(* CODESYS project canbus.20190114.1.project

Project tree, tasks and I/O mapping:
  Changsha_Xiangji_ARM_Cortex_A9_xilinx_zynq7000_linux : Changsha Xiangji-ARM Cortex A9(xilinx zynq7000)-linux, Changsha Xiangji Hiden Technology Co.Ltd, version 3.5.10.40
    application Application
      libraries: CAA Types Extern, 3.5.10.0 (CAA Technical Workgroup); VisuDialogs, * (System); CAA Real Time Clock Extern, 3.5.10.0 (CAA Technical Workgroup); CAA Callback Extern, 3.5.11.0 (CAA Technical Workgroup); CAA Can Low Level Extern, 3.5.11.0 (CAA Technical Workgroup); CAA Can Low Level Imp Extern, 3.5.11.0 (CAA Technical Workgroup); SysMem, 3.5.12.0 (System); CAA Net Base Services, 3.5.12.0 (CAA Technical Workgroup); Standard, 3.5.12.0 (System); CAA SerialCom, 3.5.12.0 (CAA Technical Workgroup); CAA File, 3.5.12.0 (CAA Technical Workgroup); CAA DTUtil Extern, 3.5.12.0 (CAA Technical Workgroup); SysFile, 3.5.9.0 (System); SysTypes2 Interfaces, * (System)
      task VISU_TASK (cyclic, interval 100 ms, priority 31) calls VisuElems.Visu_Prg
      task task_can (cyclic, interval 50 ms, priority 5) calls prg_can0, prg_can1, prg_test_can
      CAN_COMM/
        program prg_can0 [ST]
        function CAN_Send_MSG [ST]
        program prg_can1 [ST]: can1_get_data1, can1_get_data3, can1_get_data2, can1_set_send_buf
        program prg_test_can [ST]
      visualisation main
      funcs/
    SoftMotion General Axis Pool
    IoDrvMIC7001 : IoDrvMIC7001, Cyber-MI, version 18.11.1
        unmapped channels: Ai00@C16, Ai01@C28, Ai02@C17, Ai03@C29, Ai04@C30, Ai05@C19, Ai06@C31, Ai07@C20, Ai08@C18, Ai09@D18, Ai10@D20, Ai11@D31, Ai12@D19, Ai13@D30, Ai14@D29, Ai15@D17, Ai16@D28, Ai17@D16, Ai18-Do00@C25, Ai19-Do01@C24, Ai20-Do02@C13, Ai21-Do03@C01, Ai22-Do04@C03, Ai23-Do05@C04, Ai24-Do06@C05, Ai25-Do07@C06, Ai26-Do08@C08, Ai27-Do09@C09, Ai28-Do10@C10, Ai29-Do11@C11, Ai30-Do12@D34, Ai31-Do13@D35, Ai32-Do14@D23, Ai33-Do15@D12, Ai34-Do16@D10, Ai35-Do17@D09, Ai36-Do18@D08, Ai37-Do19@D07, Ai38-Do20@D05, Ai39-Do21@D04,
          Ai40-Do22@D03, Ai41-Do23@D02, Ai42-Do24@C23, Ai43-Do25@C35, Ai44-Do26@D24, Ai45-Do27@D13, Ai46-Ao00@C22, Ai47-Ao01@D14, Ai48_Pi02, Ai49_Out5V, Ai50_VCC, Ai51_VCC_L, Ai52_VCC_R, Ai53_Pwm-i0, Ai54_Pwm-i1, Ai55_Pwm-i2, Ai56_Pwm-i3, Ai57_CPU-T, Ai58_G-x, Ai59_G-y, Ai60_G-z, Ai61-reserved, Ai62-IO-cntr, Ai63-CDS-cntr, Di00-Ai00@C16, Di01-Ai01@C28, Di02-Ai02@C17, Di03-Ai03@C29, Di04-Ai04@C30, Di05-Ai05@C19, Di06-Ai06@C31, Di07-Ai07@C20, Di08-Ai08@C18, Di09-Ai09@D18, Di10-Ai10@D20, Di11-Ai11@D31, Di12-Ai12@D19, Di13-Ai13@D30, Di14-Ai14@D29, Di15-Ai15@D17,
          Di16-Ai16@D28, Di17-Ai17@D16, Di18-Ai18@C25, Di19-Ai19@C24, Di20-Ai20@C13, Di21-Ai21@C01, Di22-Ai22@C03, Di23-Ai23@C04, Di24-Ai24@C05, Di25-Ai25@C06, Di26-Ai26@C08, Di27-Ai27@C09, Di28-Ai28@C10, Di29-Ai29@C11, Di30-Ai30@D34, Di31-Ai31@D35, Di32-Ai32@D23, Di33-Ai33@D12, Di34-Ai34@D10, Di35-Ai35@D09, Di36-Ai36@D08, Di37-Ai37@D07, Di38-Ai38@D05, Di39-Ai39@D04, Di40-Ai40@D03, Di41-Ai41@D02, Di42-Ai42@C23, Di43-Ai43@C35, Di44-Ai44@D24, Di45-Ai45@D13, Di46-Ai46@C22, Di47-Ai47@D14, Di48-Pi00@C15, Di49-Pi01@C14, Di50-Pi02@D22, Di51-Pi03@D21, Di52-reserved, Di53-reserved, Di54-reserved, Di55-reserved,
          Di56-reserved, Di57-reserved, Di58-reserved, Di59-reserved, Di60-reserved, Di61-reserved, Di62-reserved, Di63-reserved, Pi00-Di48@C15, Pi01-Di49@C14, Pi02-Di50@D22, Pi03-Di51@D21, Do00-Ai18@C25, Do01-Ai19@C24, Do02-Ai20@C13, Do03-Ai21@C01, Do04-Ai22@C03, Do05-Ai23@C04, Do06-Ai24@C05, Do07-Ai25@C06, Do08-Ai26@C08, Do09-Ai27@C09, Do10-Ai28@C10, Do11-Ai29@C11, Do12-Ai30@D34, Do13-Ai31@D35, Do14-Ai32@D23, Do15-Ai33@D12, Do16-Ai34@D10, Do17-Ai35@D09, Do18-Ai36@D08, Do19-Ai37@D07, Do20-Ai38@D05, Do21-Ai39@D04, Do22-Ai40@D03, Do23-Ai41@D02, Do24-Ai42@C23, Do25-Ai43@C35, Do26-Ai44@D24, Do27-Ai45@D13,
          Do28-Pwmi00@C33, Do29-Pwmi01@C34, Do30-Pwmi02@D25, Do31-Pwmi03@D26, PWM00@C25, PWM01@C24, PWM02@C13, PWM03@C01, PWM04@C03, PWM05@C04, PWM06@C05, PWM07@C06, PWM08@C08, PWM09@C09, PWM10@C10, PWM11@C11, PWM12@D34, PWM13@D35, PWM14@D23, PWM15@D12, PWM16@D10, PWM17@D09, PWM18@D08, PWM19@D07, PWM20@D05, PWM21@D04, PWM22@D03, PWM23@D02, PWM24@C23, PWM25@C35, PWM26@D24, PWM27@D13, PWM28-Pwmi00@C33, PWM29-Pwmi01@C34, PWM30-Pwmi02@D25, PWM31-Pwmi03@D26, PWM_I_0@C33, PWM_I_1@C34, PWM_I_2@D25, PWM_I_3@D26,
          Ao00-Ai46@C22, Ao01-Ai47@D14, LED_run, LED_err, LED_usr, ctrl_ai_raw, ctrl_adjust, ctrl_adj0, ctrl_adj1, ctrl_adj2, ctrl_adj3, ctrl_adj4
    EtherCAT_Master : EtherCAT Master, 3S - Smart Software Solutions GmbH, version 3.5.12.40
        settings: NetworkName = 'eth0'; NetworkName = "eth0"; SelectNetworkByName = True; SrcAddress1 = 8719; SrcAddress2 = 3785618642
      MIR3501 : MIR3501, Cyber-MI, order no. MIR3501, version Revision=16#00000000
          settings: CheckProductID = False; CheckVendorID = False; StationAlias = 1001; Optional = False; DeviceIdenticationADO = 0; DeviceIdenticationMode = 0; DC sync0 cycletime = 4000; DC sync1 cycletime = 4000; RxTxPdo.NumberofExcludes = 0; RxTxPdo.NumberofEntries = 24; RxTxPdo.Index = 16#1600; RxTxPdo.Fixed = True; RxTxPdo.Mandatory = True; RxTxPdo.Virtual = False; RxTxPdo.Sm = 2; RxTxPdo.Su = 2; RxTxPdo.Name = 'OUT_GENERIC process data mapping'; RxTxPdo.DependOnSlot = False; RxTxPdo.DependOnSlotGroup = False; RxTxPdo.OverwrittenByModule = False; DO-00-C01.Index = 16#7000; DO-00-C01.SubIndex = 1; DO-00-C01.Size = 1; DO-00-C01.Offset = 0; DO-00-C01.DependOnSlot = False; DO-00-C01.DependOnSlotGroup = False; DO-01-C02.Index = 16#7000; DO-01-C02.SubIndex = 2; DO-01-C02.Size = 1; DO-01-C02.Offset = 0; DO-01-C02.DependOnSlot = False; DO-01-C02.DependOnSlotGroup = False; DO-02-C03.Index = 16#7000; DO-02-C03.SubIndex = 3; DO-02-C03.Size = 1; DO-02-C03.Offset = 0; DO-02-C03.DependOnSlot = False; DO-02-C03.DependOnSlotGroup = False; DO-03-C04.Index = 16#7000; DO-03-C04.SubIndex = 4;
            DO-03-C04.Size = 1; DO-03-C04.Offset = 0; DO-03-C04.DependOnSlot = False; DO-03-C04.DependOnSlotGroup = False; DO-04-C05.Index = 16#7000; DO-04-C05.SubIndex = 5; DO-04-C05.Size = 1; DO-04-C05.Offset = 0; DO-04-C05.DependOnSlot = False; DO-04-C05.DependOnSlotGroup = False; DO-05-C06.Index = 16#7000; DO-05-C06.SubIndex = 6; DO-05-C06.Size = 1; DO-05-C06.Offset = 0; DO-05-C06.DependOnSlot = False; DO-05-C06.DependOnSlotGroup = False; DO-06-C07.Index = 16#7000; DO-06-C07.SubIndex = 7; DO-06-C07.Size = 1; DO-06-C07.Offset = 0; DO-06-C07.DependOnSlot = False; DO-06-C07.DependOnSlotGroup = False; DO-07-C08.Index = 16#7000; DO-07-C08.SubIndex = 8; DO-07-C08.Size = 1; DO-07-C08.Offset = 0; DO-07-C08.DependOnSlot = False; DO-07-C08.DependOnSlotGroup = False; DO-08-C09.Index = 16#7000; DO-08-C09.SubIndex = 9; DO-08-C09.Size = 1; DO-08-C09.Offset = 0; DO-08-C09.DependOnSlot = False; DO-08-C09.DependOnSlotGroup = False; DO-09-C10.Index = 16#7000; DO-09-C10.SubIndex = 10; DO-09-C10.Size = 1; DO-09-C10.Offset = 0; DO-09-C10.DependOnSlot = False; DO-09-C10.DependOnSlotGroup = False;
            DO-10-C11.Index = 16#7000; DO-10-C11.SubIndex = 11; DO-10-C11.Size = 1; DO-10-C11.Offset = 0; DO-10-C11.DependOnSlot = False; DO-10-C11.DependOnSlotGroup = False; DO-11-C12.Index = 16#7000; DO-11-C12.SubIndex = 12; DO-11-C12.Size = 1; DO-11-C12.Offset = 0; DO-11-C12.DependOnSlot = False; DO-11-C12.DependOnSlotGroup = False; DO-12-C26.Index = 16#7000; DO-12-C26.SubIndex = 13; DO-12-C26.Size = 1; DO-12-C26.Offset = 0; DO-12-C26.DependOnSlot = False; DO-12-C26.DependOnSlotGroup = False; DO-13-C25.Index = 16#7000; DO-13-C25.SubIndex = 14; DO-13-C25.Size = 1; DO-13-C25.Offset = 0; DO-13-C25.DependOnSlot = False; DO-13-C25.DependOnSlotGroup = False; DO-14-C34.Index = 16#7000; DO-14-C34.SubIndex = 15; DO-14-C34.Size = 1; DO-14-C34.Offset = 0; DO-14-C34.DependOnSlot = False; DO-14-C34.DependOnSlotGroup = False; DO-15-C33.Index = 16#7000; DO-15-C33.SubIndex = 16; DO-15-C33.Size = 1; DO-15-C33.Offset = 0; DO-15-C33.DependOnSlot = False; DO-15-C33.DependOnSlotGroup = False; PWM-00-C26.Index = 16#7000; PWM-00-C26.SubIndex = 17; PWM-00-C26.Size = 16; PWM-00-C26.Offset = 0;
            PWM-00-C26.DependOnSlot = False; PWM-00-C26.DependOnSlotGroup = False; PWM-01-C25.Index = 16#7000; PWM-01-C25.SubIndex = 18; PWM-01-C25.Size = 16; PWM-01-C25.Offset = 0; PWM-01-C25.DependOnSlot = False; PWM-01-C25.DependOnSlotGroup = False; PWM-02-C34.Index = 16#7000; PWM-02-C34.SubIndex = 19; PWM-02-C34.Size = 16; PWM-02-C34.Offset = 0; PWM-02-C34.DependOnSlot = False; PWM-02-C34.DependOnSlotGroup = False; PWM-03-C33.Index = 16#7000; PWM-03-C33.SubIndex = 20; PWM-03-C33.Size = 16; PWM-03-C33.Offset = 0; PWM-03-C33.DependOnSlot = False; PWM-03-C33.DependOnSlotGroup = False; PWMi-00-C26.Index = 16#7000; PWMi-00-C26.SubIndex = 21; PWMi-00-C26.Size = 16; PWMi-00-C26.Offset = 0; PWMi-00-C26.DependOnSlot = False; PWMi-00-C26.DependOnSlotGroup = False; PWMi-01-C25.Index = 16#7000; PWMi-01-C25.SubIndex = 22; PWMi-01-C25.Size = 16; PWMi-01-C25.Offset = 0; PWMi-01-C25.DependOnSlot = False; PWMi-01-C25.DependOnSlotGroup = False; PWMi-02-C34.Index = 16#7000; PWMi-02-C34.SubIndex = 23; PWMi-02-C34.Size = 16; PWMi-02-C34.Offset = 0; PWMi-02-C34.DependOnSlot = False; PWMi-02-C34.DependOnSlotGroup = False; PWMi-03-C33.Index = 16#7000; PWMi-03-C33.SubIndex = 24;
            PWMi-03-C33.Size = 16; PWMi-03-C33.Offset = 0; PWMi-03-C33.DependOnSlot = False; PWMi-03-C33.DependOnSlotGroup = False; RxTxPdo.NumberofExcludes = 0; RxTxPdo.NumberofEntries = 60; RxTxPdo.Index = 16#1A00; RxTxPdo.Fixed = True; RxTxPdo.Mandatory = True; RxTxPdo.Virtual = False; RxTxPdo.Sm = 3; RxTxPdo.Su = 3; RxTxPdo.Name = 'IN_GENERIC process data mapping'; RxTxPdo.DependOnSlot = False; RxTxPdo.DependOnSlotGroup = False; RxTxPdo.OverwrittenByModule = False; AI-00-C17.Index = 16#6000; AI-00-C17.SubIndex = 1; AI-00-C17.Size = 16; AI-00-C17.Offset = 0; AI-00-C17.DependOnSlot = False; AI-00-C17.DependOnSlotGroup = False; AI-01-C29.Index = 16#6000; AI-01-C29.SubIndex = 2; AI-01-C29.Size = 16; AI-01-C29.Offset = 0; AI-01-C29.DependOnSlot = False; AI-01-C29.DependOnSlotGroup = False; AI-02-C18.Index = 16#6000; AI-02-C18.SubIndex = 3; AI-02-C18.Size = 16; AI-02-C18.Offset = 0; AI-02-C18.DependOnSlot = False; AI-02-C18.DependOnSlotGroup = False; AI-03-C30.Index = 16#6000; AI-03-C30.SubIndex = 4; AI-03-C30.Size = 16; AI-03-C30.Offset = 0; AI-03-C30.DependOnSlot = False; AI-03-C30.DependOnSlotGroup = False;
            AI-04-C14.Index = 16#6000; AI-04-C14.SubIndex = 5; AI-04-C14.Size = 16; AI-04-C14.Offset = 0; AI-04-C14.DependOnSlot = False; AI-04-C14.DependOnSlotGroup = False; AI-05-C15.Index = 16#6000; AI-05-C15.SubIndex = 6; AI-05-C15.Size = 16; AI-05-C15.Offset = 0; AI-05-C15.DependOnSlot = False; AI-05-C15.DependOnSlotGroup = False; AI-06-C21.Index = 16#6000; AI-06-C21.SubIndex = 7; AI-06-C21.Size = 16; AI-06-C21.Offset = 0; AI-06-C21.DependOnSlot = False; AI-06-C21.DependOnSlotGroup = False; AI-07-C22.Index = 16#6000; AI-07-C22.SubIndex = 8; AI-07-C22.Size = 16; AI-07-C22.Offset = 0; AI-07-C22.DependOnSlot = False; AI-07-C22.DependOnSlotGroup = False; AI-08-C01.Index = 16#6000; AI-08-C01.SubIndex = 9; AI-08-C01.Size = 16; AI-08-C01.Offset = 0; AI-08-C01.DependOnSlot = False; AI-08-C01.DependOnSlotGroup = False; AI-09-C02.Index = 16#6000; AI-09-C02.SubIndex = 10; AI-09-C02.Size = 16; AI-09-C02.Offset = 0; AI-09-C02.DependOnSlot = False; AI-09-C02.DependOnSlotGroup = False; AI-10-C03.Index = 16#6000; AI-10-C03.SubIndex = 11; AI-10-C03.Size = 16; AI-10-C03.Offset = 0;
            AI-10-C03.DependOnSlot = False; AI-10-C03.DependOnSlotGroup = False; AI-11-C04.Index = 16#6000; AI-11-C04.SubIndex = 12; AI-11-C04.Size = 16; AI-11-C04.Offset = 0; AI-11-C04.DependOnSlot = False; AI-11-C04.DependOnSlotGroup = False; AI-12-C05.Index = 16#6000; AI-12-C05.SubIndex = 13; AI-12-C05.Size = 16; AI-12-C05.Offset = 0; AI-12-C05.DependOnSlot = False; AI-12-C05.DependOnSlotGroup = False; AI-13-C06.Index = 16#6000; AI-13-C06.SubIndex = 14; AI-13-C06.Size = 16; AI-13-C06.Offset = 0; AI-13-C06.DependOnSlot = False; AI-13-C06.DependOnSlotGroup = False; AI-14-C07.Index = 16#6000; AI-14-C07.SubIndex = 15; AI-14-C07.Size = 16; AI-14-C07.Offset = 0; AI-14-C07.DependOnSlot = False; AI-14-C07.DependOnSlotGroup = False; AI-15-C08.Index = 16#6000; AI-15-C08.SubIndex = 16; AI-15-C08.Size = 16; AI-15-C08.Offset = 0; AI-15-C08.DependOnSlot = False; AI-15-C08.DependOnSlotGroup = False; AI-16-C09.Index = 16#6000; AI-16-C09.SubIndex = 17; AI-16-C09.Size = 16; AI-16-C09.Offset = 0; AI-16-C09.DependOnSlot = False; AI-16-C09.DependOnSlotGroup = False; AI-17-C10.Index = 16#6000; AI-17-C10.SubIndex = 18;
            AI-17-C10.Size = 16; AI-17-C10.Offset = 0; AI-17-C10.DependOnSlot = False; AI-17-C10.DependOnSlotGroup = False; AI-18-C11.Index = 16#6000; AI-18-C11.SubIndex = 19; AI-18-C11.Size = 16; AI-18-C11.Offset = 0; AI-18-C11.DependOnSlot = False; AI-18-C11.DependOnSlotGroup = False; AI-19-C12.Index = 16#6000; AI-19-C12.SubIndex = 20; AI-19-C12.Size = 16; AI-19-C12.Offset = 0; AI-19-C12.DependOnSlot = False; AI-19-C12.DependOnSlotGroup = False; AI-20.Index = 16#6000; AI-20.SubIndex = 21; AI-20.Size = 16; AI-20.Offset = 0; AI-20.DependOnSlot = False; AI-20.DependOnSlotGroup = False; AI-21.Index = 16#6000; AI-21.SubIndex = 22; AI-21.Size = 16; AI-21.Offset = 0; AI-21.DependOnSlot = False; AI-21.DependOnSlotGroup = False; AI-22.Index = 16#6000; AI-22.SubIndex = 23; AI-22.Size = 16; AI-22.Offset = 0; AI-22.DependOnSlot = False; AI-22.DependOnSlotGroup = False; AI-23.Index = 16#6000; AI-23.SubIndex = 24; AI-23.Size = 16; AI-23.Offset = 0; AI-23.DependOnSlot = False; AI-23.DependOnSlotGroup = False;
            DI-00-C17.Index = 16#6000; DI-00-C17.SubIndex = 25; DI-00-C17.Size = 1; DI-00-C17.Offset = 0; DI-00-C17.DependOnSlot = False; DI-00-C17.DependOnSlotGroup = False; DI-01-C29.Index = 16#6000; DI-01-C29.SubIndex = 26; DI-01-C29.Size = 1; DI-01-C29.Offset = 0; DI-01-C29.DependOnSlot = False; DI-01-C29.DependOnSlotGroup = False; DI-02-C18.Index = 16#6000; DI-02-C18.SubIndex = 27; DI-02-C18.Size = 1; DI-02-C18.Offset = 0; DI-02-C18.DependOnSlot = False; DI-02-C18.DependOnSlotGroup = False; DI-03-C30.Index = 16#6000; DI-03-C30.SubIndex = 28; DI-03-C30.Size = 1; DI-03-C30.Offset = 0; DI-03-C30.DependOnSlot = False; DI-03-C30.DependOnSlotGroup = False; DI-04-C14.Index = 16#6000; DI-04-C14.SubIndex = 29; DI-04-C14.Size = 1; DI-04-C14.Offset = 0; DI-04-C14.DependOnSlot = False; DI-04-C14.DependOnSlotGroup = False; DI-05-C15.Index = 16#6000; DI-05-C15.SubIndex = 30; DI-05-C15.Size = 1; DI-05-C15.Offset = 0; DI-05-C15.DependOnSlot = False; DI-05-C15.DependOnSlotGroup = False; DI-06-C21.Index = 16#6000; DI-06-C21.SubIndex = 31; DI-06-C21.Size = 1; DI-06-C21.Offset = 0;
            DI-06-C21.DependOnSlot = False; DI-06-C21.DependOnSlotGroup = False; DI-07-C22.Index = 16#6000; DI-07-C22.SubIndex = 32; DI-07-C22.Size = 1; DI-07-C22.Offset = 0; DI-07-C22.DependOnSlot = False; DI-07-C22.DependOnSlotGroup = False; DI-08-C01.Index = 16#6000; DI-08-C01.SubIndex = 33; DI-08-C01.Size = 1; DI-08-C01.Offset = 0; DI-08-C01.DependOnSlot = False; DI-08-C01.DependOnSlotGroup = False; DI-09-C02.Index = 16#6000; DI-09-C02.SubIndex = 34; DI-09-C02.Size = 1; DI-09-C02.Offset = 0; DI-09-C02.DependOnSlot = False; DI-09-C02.DependOnSlotGroup = False; DI-10-C03.Index = 16#6000; DI-10-C03.SubIndex = 35; DI-10-C03.Size = 1; DI-10-C03.Offset = 0; DI-10-C03.DependOnSlot = False; DI-10-C03.DependOnSlotGroup = False; DI-11-C04.Index = 16#6000; DI-11-C04.SubIndex = 36; DI-11-C04.Size = 1; DI-11-C04.Offset = 0; DI-11-C04.DependOnSlot = False; DI-11-C04.DependOnSlotGroup = False; DI-12-C05.Index = 16#6000; DI-12-C05.SubIndex = 37; DI-12-C05.Size = 1; DI-12-C05.Offset = 0; DI-12-C05.DependOnSlot = False; DI-12-C05.DependOnSlotGroup = False; DI-13-C06.Index = 16#6000; DI-13-C06.SubIndex = 38;
            DI-13-C06.Size = 1; DI-13-C06.Offset = 0; DI-13-C06.DependOnSlot = False; DI-13-C06.DependOnSlotGroup = False; DI-14-C07.Index = 16#6000; DI-14-C07.SubIndex = 39; DI-14-C07.Size = 1; DI-14-C07.Offset = 0; DI-14-C07.DependOnSlot = False; DI-14-C07.DependOnSlotGroup = False; DI-15-C08.Index = 16#6000; DI-15-C08.SubIndex = 40; DI-15-C08.Size = 1; DI-15-C08.Offset = 0; DI-15-C08.DependOnSlot = False; DI-15-C08.DependOnSlotGroup = False; DI-16-C09.Index = 16#6000; DI-16-C09.SubIndex = 41; DI-16-C09.Size = 1; DI-16-C09.Offset = 0; DI-16-C09.DependOnSlot = False; DI-16-C09.DependOnSlotGroup = False; DI-17-C10.Index = 16#6000; DI-17-C10.SubIndex = 42; DI-17-C10.Size = 1; DI-17-C10.Offset = 0; DI-17-C10.DependOnSlot = False; DI-17-C10.DependOnSlotGroup = False; DI-18-C11.Index = 16#6000; DI-18-C11.SubIndex = 43; DI-18-C11.Size = 1; DI-18-C11.Offset = 0; DI-18-C11.DependOnSlot = False; DI-18-C11.DependOnSlotGroup = False; DI-19-C12.Index = 16#6000; DI-19-C12.SubIndex = 44; DI-19-C12.Size = 1; DI-19-C12.Offset = 0; DI-19-C12.DependOnSlot = False; DI-19-C12.DependOnSlotGroup = False;
            DI-20-C27.Index = 16#6000; DI-20-C27.SubIndex = 45; DI-20-C27.Size = 1; DI-20-C27.Offset = 0; DI-20-C27.DependOnSlot = False; DI-20-C27.DependOnSlotGroup = False; DI-21-C16.Index = 16#6000; DI-21-C16.SubIndex = 46; DI-21-C16.Size = 1; DI-21-C16.Offset = 0; DI-21-C16.DependOnSlot = False; DI-21-C16.DependOnSlotGroup = False; DI-22-C19.Index = 16#6000; DI-22-C19.SubIndex = 47; DI-22-C19.Size = 1; DI-22-C19.Offset = 0; DI-22-C19.DependOnSlot = False; DI-22-C19.DependOnSlotGroup = False; DI-23-C20.Index = 16#6000; DI-23-C20.SubIndex = 48; DI-23-C20.Size = 1; DI-23-C20.Offset = 0; DI-23-C20.DependOnSlot = False; DI-23-C20.DependOnSlotGroup = False; DI-24.Index = 16#6000; DI-24.SubIndex = 49; DI-24.Size = 1; DI-24.Offset = 0; DI-24.DependOnSlot = False; DI-24.DependOnSlotGroup = False; DI-25.Index = 16#6000; DI-25.SubIndex = 50; DI-25.Size = 1; DI-25.Offset = 0; DI-25.DependOnSlot = False; DI-25.DependOnSlotGroup = False; DI-26.Index = 16#6000; DI-26.SubIndex = 51; DI-26.Size = 1; DI-26.Offset = 0;
            DI-26.DependOnSlot = False; DI-26.DependOnSlotGroup = False; DI-27.Index = 16#6000; DI-27.SubIndex = 52; DI-27.Size = 1; DI-27.Offset = 0; DI-27.DependOnSlot = False; DI-27.DependOnSlotGroup = False; DI-28.Index = 16#6000; DI-28.SubIndex = 53; DI-28.Size = 1; DI-28.Offset = 0; DI-28.DependOnSlot = False; DI-28.DependOnSlotGroup = False; DI-29.Index = 16#6000; DI-29.SubIndex = 54; DI-29.Size = 1; DI-29.Offset = 0; DI-29.DependOnSlot = False; DI-29.DependOnSlotGroup = False; DI-30.Index = 16#6000; DI-30.SubIndex = 55; DI-30.Size = 1; DI-30.Offset = 0; DI-30.DependOnSlot = False; DI-30.DependOnSlotGroup = False; DI-31.Index = 16#6000; DI-31.SubIndex = 56; DI-31.Size = 1; DI-31.Offset = 0; DI-31.DependOnSlot = False; DI-31.DependOnSlotGroup = False; PI-00-C27.Index = 16#6000; PI-00-C27.SubIndex = 57; PI-00-C27.Size = 16; PI-00-C27.Offset = 0; PI-00-C27.DependOnSlot = False; PI-00-C27.DependOnSlotGroup = False; PI-01-C16.Index = 16#6000; PI-01-C16.SubIndex = 58;
            PI-01-C16.Size = 16; PI-01-C16.Offset = 0; PI-01-C16.DependOnSlot = False; PI-01-C16.DependOnSlotGroup = False; PI-02-C19.Index = 16#6000; PI-02-C19.SubIndex = 59; PI-02-C19.Size = 16; PI-02-C19.Offset = 0; PI-02-C19.DependOnSlot = False; PI-02-C19.DependOnSlotGroup = False; PI-03-C20.Index = 16#6000; PI-03-C20.SubIndex = 60; PI-03-C20.Size = 16; PI-03-C20.Offset = 0; PI-03-C20.DependOnSlot = False; PI-03-C20.DependOnSlotGroup = False; DO-00-C01.Name = 'DO-00-C01'; DO-00-C01.DataType = 'BIT'; DO-00-C01.Default = ''; DO-00-C01.Comment = ''; DO-01-C02.Name = 'DO-01-C02'; DO-01-C02.DataType = 'BIT'; DO-01-C02.Default = ''; DO-01-C02.Comment = ''; DO-02-C03.Name = 'DO-02-C03'; DO-02-C03.DataType = 'BIT'; DO-02-C03.Default = ''; DO-02-C03.Comment = ''; DO-03-C04.Name = 'DO-03-C04'; DO-03-C04.DataType = 'BIT'; DO-03-C04.Default = ''; DO-03-C04.Comment = ''; DO-04-C05.Name = 'DO-04-C05'; DO-04-C05.DataType = 'BIT'; DO-04-C05.Default = ''; DO-04-C05.Comment = ''; DO-05-C06.Name = 'DO-05-C06'; DO-05-C06.DataType = 'BIT'; DO-05-C06.Default = ''; DO-05-C06.Comment = '';
            DO-06-C07.Name = 'DO-06-C07'; DO-06-C07.DataType = 'BIT'; DO-06-C07.Default = ''; DO-06-C07.Comment = ''; DO-07-C08.Name = 'DO-07-C08'; DO-07-C08.DataType = 'BIT'; DO-07-C08.Default = ''; DO-07-C08.Comment = ''; DO-08-C09.Name = 'DO-08-C09'; DO-08-C09.DataType = 'BIT'; DO-08-C09.Default = ''; DO-08-C09.Comment = ''; DO-09-C10.Name = 'DO-09-C10'; DO-09-C10.DataType = 'BIT'; DO-09-C10.Default = ''; DO-09-C10.Comment = ''; DO-10-C11.Name = 'DO-10-C11'; DO-10-C11.DataType = 'BIT'; DO-10-C11.Default = ''; DO-10-C11.Comment = ''; DO-11-C12.Name = 'DO-11-C12'; DO-11-C12.DataType = 'BIT'; DO-11-C12.Default = ''; DO-11-C12.Comment = ''; DO-12-C26.Name = 'DO-12-C26'; DO-12-C26.DataType = 'BIT'; DO-12-C26.Default = ''; DO-12-C26.Comment = ''; DO-13-C25.Name = 'DO-13-C25'; DO-13-C25.DataType = 'BIT'; DO-13-C25.Default = ''; DO-13-C25.Comment = ''; DO-14-C34.Name = 'DO-14-C34'; DO-14-C34.DataType = 'BIT'; DO-14-C34.Default = ''; DO-14-C34.Comment = ''; DO-15-C33.Name = 'DO-15-C33'; DO-15-C33.DataType = 'BIT'; DO-15-C33.Default = ''; DO-15-C33.Comment = '';
            PWM-00-C26.Name = 'PWM-00-C26'; PWM-00-C26.DataType = 'UINT'; PWM-00-C26.Default = ''; PWM-00-C26.Comment = ''; PWM-01-C25.Name = 'PWM-01-C25'; PWM-01-C25.DataType = 'UINT'; PWM-01-C25.Default = ''; PWM-01-C25.Comment = ''; PWM-02-C34.Name = 'PWM-02-C34'; PWM-02-C34.DataType = 'UINT'; PWM-02-C34.Default = ''; PWM-02-C34.Comment = ''; PWM-03-C33.Name = 'PWM-03-C33'; PWM-03-C33.DataType = 'UINT'; PWM-03-C33.Default = ''; PWM-03-C33.Comment = ''; PWMi-00-C26.Name = 'PWMi-00-C26'; PWMi-00-C26.DataType = 'UINT'; PWMi-00-C26.Default = ''; PWMi-00-C26.Comment = ''; PWMi-01-C25.Name = 'PWMi-01-C25'; PWMi-01-C25.DataType = 'UINT'; PWMi-01-C25.Default = ''; PWMi-01-C25.Comment = ''; PWMi-02-C34.Name = 'PWMi-02-C34'; PWMi-02-C34.DataType = 'UINT'; PWMi-02-C34.Default = ''; PWMi-02-C34.Comment = ''; PWMi-03-C33.Name = 'PWMi-03-C33'; PWMi-03-C33.DataType = 'UINT'; PWMi-03-C33.Default = ''; PWMi-03-C33.Comment = ''; AI-00-C17.Name = 'AI-00-C17'; AI-00-C17.DataType = 'UINT'; AI-00-C17.Default = ''; AI-00-C17.Comment = ''; AI-01-C29.Name = 'AI-01-C29'; AI-01-C29.DataType = 'UINT'; AI-01-C29.Default = ''; AI-01-C29.Comment = '';
            AI-02-C18.Name = 'AI-02-C18'; AI-02-C18.DataType = 'UINT'; AI-02-C18.Default = ''; AI-02-C18.Comment = ''; AI-03-C30.Name = 'AI-03-C30'; AI-03-C30.DataType = 'UINT'; AI-03-C30.Default = ''; AI-03-C30.Comment = ''; AI-04-C14.Name = 'AI-04-C14'; AI-04-C14.DataType = 'UINT'; AI-04-C14.Default = ''; AI-04-C14.Comment = ''; AI-05-C15.Name = 'AI-05-C15'; AI-05-C15.DataType = 'UINT'; AI-05-C15.Default = ''; AI-05-C15.Comment = ''; AI-06-C21.Name = 'AI-06-C21'; AI-06-C21.DataType = 'UINT'; AI-06-C21.Default = ''; AI-06-C21.Comment = ''; AI-07-C22.Name = 'AI-07-C22'; AI-07-C22.DataType = 'UINT'; AI-07-C22.Default = ''; AI-07-C22.Comment = ''; AI-08-C01.Name = 'AI-08-C01'; AI-08-C01.DataType = 'UINT'; AI-08-C01.Default = ''; AI-08-C01.Comment = ''; AI-09-C02.Name = 'AI-09-C02'; AI-09-C02.DataType = 'UINT'; AI-09-C02.Default = ''; AI-09-C02.Comment = ''; AI-10-C03.Name = 'AI-10-C03'; AI-10-C03.DataType = 'UINT'; AI-10-C03.Default = ''; AI-10-C03.Comment = ''; AI-11-C04.Name = 'AI-11-C04'; AI-11-C04.DataType = 'UINT'; AI-11-C04.Default = ''; AI-11-C04.Comment = '';
            AI-12-C05.Name = 'AI-12-C05'; AI-12-C05.DataType = 'UINT'; AI-12-C05.Default = ''; AI-12-C05.Comment = ''; AI-13-C06.Name = 'AI-13-C06'; AI-13-C06.DataType = 'UINT'; AI-13-C06.Default = ''; AI-13-C06.Comment = ''; AI-14-C07.Name = 'AI-14-C07'; AI-14-C07.DataType = 'UINT'; AI-14-C07.Default = ''; AI-14-C07.Comment = ''; AI-15-C08.Name = 'AI-15-C08'; AI-15-C08.DataType = 'UINT'; AI-15-C08.Default = ''; AI-15-C08.Comment = ''; AI-16-C09.Name = 'AI-16-C09'; AI-16-C09.DataType = 'UINT'; AI-16-C09.Default = ''; AI-16-C09.Comment = ''; AI-17-C10.Name = 'AI-17-C10'; AI-17-C10.DataType = 'UINT'; AI-17-C10.Default = ''; AI-17-C10.Comment = ''; AI-18-C11.Name = 'AI-18-C11'; AI-18-C11.DataType = 'UINT'; AI-18-C11.Default = ''; AI-18-C11.Comment = ''; AI-19-C12.Name = 'AI-19-C12'; AI-19-C12.DataType = 'UINT'; AI-19-C12.Default = ''; AI-19-C12.Comment = ''; AI-20.Name = 'AI-20'; AI-20.DataType = 'UINT'; AI-20.Default = ''; AI-20.Comment = ''; AI-21.Name = 'AI-21'; AI-21.DataType = 'UINT'; AI-21.Default = ''; AI-21.Comment = '';
            AI-22.Name = 'AI-22'; AI-22.DataType = 'UINT'; AI-22.Default = ''; AI-22.Comment = ''; AI-23.Name = 'AI-23'; AI-23.DataType = 'UINT'; AI-23.Default = ''; AI-23.Comment = ''; DI-00-C17.Name = 'DI-00-C17'; DI-00-C17.DataType = 'BIT'; DI-00-C17.Default = ''; DI-00-C17.Comment = ''; DI-01-C29.Name = 'DI-01-C29'; DI-01-C29.DataType = 'BIT'; DI-01-C29.Default = ''; DI-01-C29.Comment = ''; DI-02-C18.Name = 'DI-02-C18'; DI-02-C18.DataType = 'BIT'; DI-02-C18.Default = ''; DI-02-C18.Comment = ''; DI-03-C30.Name = 'DI-03-C30'; DI-03-C30.DataType = 'BIT'; DI-03-C30.Default = ''; DI-03-C30.Comment = ''; DI-04-C14.Name = 'DI-04-C14'; DI-04-C14.DataType = 'BIT'; DI-04-C14.Default = ''; DI-04-C14.Comment = ''; DI-05-C15.Name = 'DI-05-C15'; DI-05-C15.DataType = 'BIT'; DI-05-C15.Default = ''; DI-05-C15.Comment = ''; DI-06-C21.Name = 'DI-06-C21'; DI-06-C21.DataType = 'BIT'; DI-06-C21.Default = ''; DI-06-C21.Comment = ''; DI-07-C22.Name = 'DI-07-C22'; DI-07-C22.DataType = 'BIT'; DI-07-C22.Default = ''; DI-07-C22.Comment = '';
            DI-08-C01.Name = 'DI-08-C01'; DI-08-C01.DataType = 'BIT'; DI-08-C01.Default = ''; DI-08-C01.Comment = ''; DI-09-C02.Name = 'DI-09-C02'; DI-09-C02.DataType = 'BIT'; DI-09-C02.Default = ''; DI-09-C02.Comment = ''; DI-10-C03.Name = 'DI-10-C03'; DI-10-C03.DataType = 'BIT'; DI-10-C03.Default = ''; DI-10-C03.Comment = ''; DI-11-C04.Name = 'DI-11-C04'; DI-11-C04.DataType = 'BIT'; DI-11-C04.Default = ''; DI-11-C04.Comment = ''; DI-12-C05.Name = 'DI-12-C05'; DI-12-C05.DataType = 'BIT'; DI-12-C05.Default = ''; DI-12-C05.Comment = ''; DI-13-C06.Name = 'DI-13-C06'; DI-13-C06.DataType = 'BIT'; DI-13-C06.Default = ''; DI-13-C06.Comment = ''; DI-14-C07.Name = 'DI-14-C07'; DI-14-C07.DataType = 'BIT'; DI-14-C07.Default = ''; DI-14-C07.Comment = ''; DI-15-C08.Name = 'DI-15-C08'; DI-15-C08.DataType = 'BIT'; DI-15-C08.Default = ''; DI-15-C08.Comment = ''; DI-16-C09.Name = 'DI-16-C09'; DI-16-C09.DataType = 'BIT'; DI-16-C09.Default = ''; DI-16-C09.Comment = ''; DI-17-C10.Name = 'DI-17-C10'; DI-17-C10.DataType = 'BIT'; DI-17-C10.Default = ''; DI-17-C10.Comment = '';
            DI-18-C11.Name = 'DI-18-C11'; DI-18-C11.DataType = 'BIT'; DI-18-C11.Default = ''; DI-18-C11.Comment = ''; DI-19-C12.Name = 'DI-19-C12'; DI-19-C12.DataType = 'BIT'; DI-19-C12.Default = ''; DI-19-C12.Comment = ''; DI-20-C27.Name = 'DI-20-C27'; DI-20-C27.DataType = 'BIT'; DI-20-C27.Default = ''; DI-20-C27.Comment = ''; DI-21-C16.Name = 'DI-21-C16'; DI-21-C16.DataType = 'BIT'; DI-21-C16.Default = ''; DI-21-C16.Comment = ''; DI-22-C19.Name = 'DI-22-C19'; DI-22-C19.DataType = 'BIT'; DI-22-C19.Default = ''; DI-22-C19.Comment = ''; DI-23-C20.Name = 'DI-23-C20'; DI-23-C20.DataType = 'BIT'; DI-23-C20.Default = ''; DI-23-C20.Comment = ''; DI-24.Name = 'DI-24'; DI-24.DataType = 'BIT'; DI-24.Default = ''; DI-24.Comment = ''; DI-25.Name = 'DI-25'; DI-25.DataType = 'BIT'; DI-25.Default = ''; DI-25.Comment = ''; DI-26.Name = 'DI-26'; DI-26.DataType = 'BIT'; DI-26.Default = ''; DI-26.Comment = ''; DI-27.Name = 'DI-27'; DI-27.DataType = 'BIT'; DI-27.Default = ''; DI-27.Comment = '';
            DI-28.Name = 'DI-28'; DI-28.DataType = 'BIT'; DI-28.Default = ''; DI-28.Comment = ''; DI-29.Name = 'DI-29'; DI-29.DataType = 'BIT'; DI-29.Default = ''; DI-29.Comment = ''; DI-30.Name = 'DI-30'; DI-30.DataType = 'BIT'; DI-30.Default = ''; DI-30.Comment = ''; DI-31.Name = 'DI-31'; DI-31.DataType = 'BIT'; DI-31.Default = ''; DI-31.Comment = ''; PI-00-C27.Name = 'PI-00-C27'; PI-00-C27.DataType = 'UINT'; PI-00-C27.Default = ''; PI-00-C27.Comment = ''; PI-01-C16.Name = 'PI-01-C16'; PI-01-C16.DataType = 'UINT'; PI-01-C16.Default = ''; PI-01-C16.Comment = ''; PI-02-C19.Name = 'PI-02-C19'; PI-02-C19.DataType = 'UINT'; PI-02-C19.Default = ''; PI-02-C19.Comment = ''; PI-03-C20.Name = 'PI-03-C20'; PI-03-C20.DataType = 'UINT'; PI-03-C20.Default = ''; PI-03-C20.Comment = ''
          unmapped channels: DO-00-C01, DO-01-C02, DO-02-C03, DO-03-C04, DO-04-C05, DO-05-C06, DO-06-C07, DO-07-C08, DO-08-C09, DO-09-C10, DO-10-C11, DO-11-C12, DO-12-C26, DO-13-C25, DO-14-C34, DO-15-C33, PWM-00-C26, PWM-01-C25, PWM-02-C34, PWM-03-C33, PWMi-00-C26, PWMi-01-C25, PWMi-02-C34, PWMi-03-C33, AI-00-C17, AI-01-C29, AI-02-C18, AI-03-C30, AI-04-C14, AI-05-C15, AI-06-C21, AI-07-C22, AI-08-C01, AI-09-C02, AI-10-C03, AI-11-C04, AI-12-C05, AI-13-C06, AI-14-C07, AI-15-C08,
            AI-16-C09, AI-17-C10, AI-18-C11, AI-19-C12, AI-20, AI-21, AI-22, AI-23, DI-00-C17, DI-01-C29, DI-02-C18, DI-03-C30, DI-04-C14, DI-05-C15, DI-06-C21, DI-07-C22, DI-08-C01, DI-09-C02, DI-10-C03, DI-11-C04, DI-12-C05, DI-13-C06, DI-14-C07, DI-15-C08, DI-16-C09, DI-17-C10, DI-18-C11, DI-19-C12, DI-20-C27, DI-21-C16, DI-22-C19, DI-23-C20, DI-24, DI-25, DI-26, DI-27, DI-28, DI-29, DI-30, DI-31,
            PI-00-C27, PI-01-C16, PI-02-C19, PI-03-C20
  5ce3da45-db07-42e7-a21c-a00fff4ed8f6|C:\Users\Administrator\Desktop\robotview1.bmp
  5ce3da45-db07-42e7-a21c-a00fff4ed8f6|C:\Users\Administrator\Desktop\robotview2.bmp
  text list GlobalTextList
  5ce3da45-db07-42e7-a21c-a00fff4ed8f6|C:\Users\Administrator\Desktop\1129.bmp
  5ce3da45-db07-42e7-a21c-a00fff4ed8f6|C:\Users\Administrator\Desktop\robotview0.bmp
*)

// Changsha_Xiangji_ARM_Cortex_A9_xilinx_zynq7000_linux/Application/CAN_COMM/prg_can0
PROGRAM prg_can0   //CAN0   与底盘和显示屏通信
VAR
	hCan0:CAA.HANDLE:=0;
    CanWriteData : ARRAY[0..7] OF BYTE;
    CanWriteMsgID:UDINT;
	CanReadData : ARRAY[0..7] OF BYTE;  
	CanReadMsgID:UDINT;
	bModifyTimeFlag :BOOL := FALSE;
	
	//通过CAN总线从底盘读到的信息
	can_data_ready:BOOL := FALSE;
	can_data_speed:BYTE := 0;
	can_data_soc:BYTE := 0;
	
	//通过CAN总线从显示屏读到的信息
	c00byte0bit0_both_wash_sweep:BOOL := FALSE;
	c00byte0bit1_left_wash_sweep:BOOL := FALSE;
	c00byte0bit2_right_wash_sweep:BOOL := FALSE;
	c00byte0bit3_both_sweep:BOOL := FALSE;
	c00byte0bit4_left_sweep:BOOL := FALSE;
	c00byte0bit5_right_sweep:BOOL := FALSE;
	c00byte0bit6_both_wash:BOOL := FALSE;
	c00byte0bit7_left_wash:BOOL := FALSE;
	
	c00byte1bit0_right_wash:BOOL := FALSE;
	c00byte1bit1_stop_sweep:BOOL := FALSE;
	c00byte1bit2_start_motor:BOOL := FALSE;
	c00byte1bit3_stop_motor:BOOL := FALSE;
	c00byte1bit4_speed_add:BOOL := FALSE;
	c00byte1bit5_speed_dec:BOOL := FALSE;
	c00byte1bit6_normal_speed:BOOL := FALSE;
	c00byte1bit7_high_speed:BOOL := FALSE;
	
	c00byte2bit0_garbage_close:BOOL := FALSE;
	c00byte2bit1_garbage_open:BOOL := FALSE;
	c00byte2bit2_garbage_up:BOOL := FALSE;
	c00byte2bit3_garbage_down:BOOL := FALSE;
	c00byte2bit4_fog_bump:BOOL := FALSE;
	c00byte2bit5_selfclean:BOOL := FALSE;
	c00byte2bit6_wastewater_pump:BOOL := FALSE;
	c00byte2bit7_res :BOOL := FALSE;
	
	c00byte3bit0_sweep_high:BOOL := FALSE;
	c00byte3bit1_sweep_middle:BOOL := FALSE;
	c00byte3bit2_sweep_low:BOOL := FALSE;
	c00byte3bit3_highpress_wash:BOOL := FALSE;
	c00byte3bit4_pointshoot_up:BOOL := FALSE;
	c00byte3bit5_pointshoot_down:BOOL := FALSE;
	c00byte3bit6_pointshoot_left:BOOL := FALSE;
	c00byte3bit7_pointshoot_right:BOOL := FALSE;

	c00byte4bit0_drain_start:BOOL := FALSE;
	c00byte4bit1_drain_auto:BOOL := FALSE;
	c00byte4bit2_drain_manual:BOOL := FALSE;
	c00byte4bit3_left_drain:BOOL := FALSE;
	c00byte4bit4_right_drain:BOOL := FALSE;
	c00byte4bit5_sub_drain:BOOL := FALSE;
	c00byte4bit6_selfclean_drain:BOOL := FALSE;
	c00byte4bit7_spout_drain:BOOL := FALSE;
	
	c00byte6bit0_func_test:BOOL := FALSE;
	c00byte6bit1_change_sweeper:BOOL := FALSE;
	c00byte6bit2_intelligent:BOOL := FALSE;
	c00byte6bit3_cleanly:BOOL := FALSE;
	c00byte6bit4_normal:BOOL := FALSE;
	c00byte6bit5_dirty:BOOL := FALSE;
	
	c01byte0bit3_test_watercooler_pump:BOOL := FALSE;
	c01byte0bit4_test_cooler_fan:BOOL := FALSE;
	
	c01byte1bit0_test_sweeper_middle:BOOL := FALSE;
	c01byte1bit1_test_sweeper_low:BOOL := FALSE;
	c01byte1bit2_test_left_sweeper:BOOL := FALSE;
	c01byte1bit3_test_right_sweeper:BOOL := FALSE;
	c01byte1bit4_test_both_sweeper:BOOL := FALSE;
	c01byte1bit5_test_box_down:BOOL := FALSE;
	c01byte1bit6_test_box_up:BOOL := FALSE;
	c01byte1bit7_test_sucker_down:BOOL := FALSE;
	
	c01byte2bit0_test_sucker_up:BOOL := FALSE;
	c01byte2bit1_test_box_open:BOOL := FALSE;
	c01byte2bit2_test_box_close:BOOL := FALSE;
	
	c01byte2bit6_test_left_sweeper_down:BOOL := FALSE;
	c01byte2bit7_test_left_sweeper_up:BOOL := FALSE;
	
	c01byte3bit0_test_right_sweeper_down:BOOL := FALSE;
	c01byte3bit1_test_right_sweeper_up:BOOL := FALSE;
	c01byte3bit2_test_left_sweeper_out:BOOL := FALSE;
	c01byte3bit3_test_right_sweeper_out:BOOL := FALSE;
	c01byte3bit4_test_left_shooter_out:BOOL := FALSE;
	c01byte3bit5_test_right_shooter_out:BOOL := FALSE;
	c01byte3bit6_test_left_shooter_water:BOOL := FALSE;
	c01byte3bit7_test_right_shooter_water:BOOL := FALSE;
	
	c01byte4bit0_test_sucker_water:BOOL := FALSE;
	c01byte4bit1_test_highpress_wash:BOOL := FALSE;
	c01byte4bit2_test_selfclean:BOOL := FALSE;
	c01byte4bit3_test_highpress_pump_gearin:BOOL := FALSE;
	c01byte4bit4_test_fogpump:BOOL := FALSE;
	
	c01byte5bit2_test_wastewater_pump:BOOL := FALSE;
	c01byte5bit3_test_wastewater_valve:BOOL := FALSE;
	
	c01byte6bit0_test_backup_power:BOOL := FALSE;
	
	c02byte45_speed_change :UINT := 0;
	c02byte67_sub_motor_min_speed:UINT := 0;
	
	c03byte01_normal_speed:UINT := 0;
	c03byte23_high_speed:UINT := 0;
	c03byte45_sweeper_speed:UINT := 0;
	
	c04byte01_highpress_pump_overspeed_warning:UINT := 0;
	c04byte23_highpress_pump_overspeed_stop:UINT := 0;
	c04byte45_sub_motor_max_speed:UINT := 0;
	c04byte67_sub_motor_idle_speed:UINT := 0;
	
	//通过CAN总线发送到显示屏的信息
	s00byte0bit0_res:BOOL := FALSE;
	
	s00byte1bit0_res:BOOL := FALSE;
	s00byte1bit1_wastewater_full:BOOL := FALSE;
	s00byte1bit2_oil_filter_block:BOOL := FALSE;
	s00byte1bit3_oil_low:BOOL := FALSE;
	s00byte1bit4_res:BOOL := FALSE;
	s00byte1bit5_tank_no_water:BOOL := FALSE;
	s00byte1bit6_res:BOOL := FALSE;
	s00byte1bit7_back_error_stop:BOOL := FALSE;
	
	s00byte2bit0_wastewater_full_stop:BOOL := FALSE;
	s00byte2bit1_electronic_power_fault:BOOL := FALSE;
	s00byte2bit2_highpress_pump_overspeed_warning:BOOL := FALSE;
	s00byte2bit3_highpress_pump_overspeed_stop:BOOL := FALSE;
	s00byte2bit4_please_close_test:BOOL := FALSE;
	s00byte2bit5_being_back:BOOL := FALSE;
	s00byte2bit6_please_open_motor:BOOL := FALSE;
	s00byte2bit7_please_open_test:BOOL := FALSE;
	
	s00byte3bit0_air_press_low:BOOL := FALSE;
	s00byte3bit1_back_the_truck:BOOL := FALSE;
	s00byte3bit2_res:BOOL := FALSE;
	s00byte3bit3_highpress_pump_not_gearin:BOOL := FALSE;
	s00byte3bit4_water_valve_not_on:BOOL := FALSE;
	s00byte3bit5_highpress_blow_valve_not_on:BOOL := FALSE;
	s00byte3bit6_highpress_water_valve_not_on:BOOL := FALSE;
	s00byte3bit7_please_open_box_door:BOOL := FALSE;
	
	s00byte4bit0_pump_valve_not_no:BOOL := FALSE;
	s00byte4bit1_pump_press_fault:BOOL := FALSE;
	s00byte4bit2_fault_stop:BOOL := FALSE;
	s00byte4bit3_please_putdown_supporter:BOOL := FALSE;
	
	s00byte4bit6_chassis_can_fault:BOOL := FALSE;
	s00byte4bit7_motordriver_can_fault:BOOL :=FALSE;
	
	s00byte5bit0_sub_wastebox_error:BOOL := FALSE;
	s00byte5bit1_sub1_wastebox_full:BOOL := FALSE;
	s00byte5bit2_sub2_wastebox_full:BOOL := FALSE;
	s00byte5bit3_water_release_valve_not_close:BOOL := FALSE;
	s00byte5bit4_water_release_valve_not_copen:BOOL := FALSE;
	s00byte5bit5_backup_power_on:BOOL := FALSE;
	s00byte5bit6_power_low_20percent:BOOL := FALSE;
	s00byte5bit7_chassis_no_high_voltage:BOOL := FALSE;
	
	s00byte6bit0_get_power_switch:BOOL := FALSE;
	s00byte6bit1_highpress_water_valve_on:BOOL := FALSE;
	s00byte6bit2_box_door_close:BOOL := FALSE;
	s00byte6bit3_highpress_blow_valve_on:BOOL := FALSE;
	s00byte6bit4_air_press_low:BOOL := FALSE;
	s00byte6bit5_wastewater_full:BOOL := FALSE;
	s00byte6bit6_left_supporter_down:BOOL := FALSE;
	s00byte6bit7_right_supporter_down:BOOL := FALSE;
	
	s00byte7bit4_fog_pump_press_ok:BOOL := FALSE;
	s00byte7bit5_oil_level_low:BOOL := FALSE;
	s00byte7bit6_oil_filter_block:BOOL := FALSE;
	
	s01byte0bit0_power_on:BOOL := FALSE;
	s01byte0bit1_back_the_truck:BOOL := FALSE;
	s01byte0bit2_res:BOOL := FALSE;
	s01byte0bit3_cleanwater_low:BOOL := FALSE;
	
	s01byte1bit0_box_down:BOOL := FALSE;
	s01byte1bit1_box_up:BOOL := FALSE;
	s01byte1bit2_sucker_down:BOOL := FALSE;
	s01byte1bit3_sucker_up:BOOL := FALSE;
	s01byte1bit4_boxdoor_close:BOOL := FALSE;
	s01byte1bit5_boxdoor_open:BOOL := FALSE;
	s01byte1bit6_left_sweeper_up:BOOL := FALSE;
	s01byte1bit7_left_sweeper_down:BOOL := FALSE;
	
	s01byte2bit0_right_sweeper_up:BOOL := FALSE;
	s01byte2bit1_right_sweeper_down:BOOL := FALSE;
	s01byte2bit2_cleanwater_high:BOOL := FALSE;
	s01byte2bit3_alterable_box_low:BOOL := FALSE;
	s01byte2bit4_res:BOOL := FALSE;
	
	s01byte3bit3_right_shooter_out:BOOL := FALSE;
	s01byte3bit4_left_shooter_out:BOOL := FALSE;
	s01byte3bit5_waterpump_gearin:BOOL := FALSE;
	s01byte3bit6_left_shooter_water:BOOL := FALSE;
	s01byte3bit7_right_shooter_water:BOOL := FALSE;
	
	s01byte4bit0_sucker_shooter_water:BOOL := FALSE;
	s01byte4bit1_selfclean_shooter_water:BOOL := FALSE;
	s01byte4bit2_high_sub_shooter_water:BOOL := FALSE;
	s01byte4bit3_water_release_valve:BOOL := FALSE;
	s01byte4bit4_oil_release_valve:BOOL := FALSE;
	s01byte4bit5_sweeper_middle_speed:BOOL := FALSE;
	s01byte4bit6_sweeper_low_speed:BOOL := FALSE;
	s01byte4bit7_left_sweeper_back:BOOL := FALSE;
	
	s01byte5bit0_left_sweeper_down:BOOL := FALSE;
	s01byte5bit1_right_sweeper_back:BOOL := FALSE;
	s01byte5bit2_right_sweeper_down:BOOL := FALSE;
	s01byte5bit3_left_all_sweep:BOOL := FALSE;
	s01byte5bit5_right_sweep:BOOL := FALSE;
	
	s01byte6bit0_right_all_sweep:BOOL := FALSE;
	s01byte6bit1_box_down:BOOL := FALSE;
	s01byte6bit2_box_up:BOOL := FALSE;
	s01byte6bit3_sucker_up:BOOL := FALSE;
	s01byte6bit4_sucker_down:BOOL := FALSE;
	s01byte6bit5_boxdoor_close:BOOL := FALSE;
	s01byte6bit6_boxdoor_open:BOOL := FALSE;
	s01byte6bit7_cleanwater_pump:BOOL := FALSE;
	
	s01byte7bit1_cooler_pump_motor:BOOL := FALSE;
	s01byte7bit2_cooler_fan:BOOL := FALSE;
	s01byte7bit3_fog_pump:BOOL := FALSE;
	
	s02byte0bit67_right_shooter_out:BYTE := 0;
	
	s02byte1bit01_left_shooter_out:BYTE := 0;
	s02byte1bit23_waterpump_gearin:BYTE := 0;
	s02byte1bit45_left_shooter_valve_open:BYTE := 0;
	s02byte1bit67_right_shooter_valve_open:BYTE := 0;
	
	s02byte2bit01_sucker_shooter_valve_open:BYTE := 0;
	s02byte2bit23_selfclean_shooter_valve_open:BYTE := 0;
	s02byte2bit45_high_sub_shooter_valve_open:BYTE := 0;
	s02byte2bit67_water_release_valve:BYTE := 0;
	
	s02byte3bit01_oil_release_valve:BYTE := 0;
	s02byte3bit23_sweeper_middle_speed:BYTE := 0;
	s02byte3bit45_sweeper_low_speed:BYTE := 0;
	s02byte3bit67_left_sweeper_back:BYTE := 0;
	
	s02byte4bit01_left_sweeper_down:BYTE := 0;
	s02byte4bit23_right_sweeper_back:BYTE := 0;
	s02byte4bit45_right_sweeper_down:BYTE := 0;
	s02byte4bit67_left_all_sweep:BYTE := 0;
	
	s02byte5bit01_right_sweep:BYTE := 0;
	s02byte5bit23_res:BYTE := 0;
	
	s02byte6bit01_right_all_sweep:BYTE := 0;
	s02byte6bit23_box_down:BYTE := 0;
	s02byte6bit45_box_up:BYTE := 0;
	s02byte6bit67_sucker_up:BYTE := 0;
	
	s02byte7bit01_sucker_down:BYTE := 0;
	s02byte7bit23_boxdoor_close:BYTE := 0;
	s02byte7bit45_boxdoor_open:BYTE := 0;
	s02byte7bit67_cleanwater_pump:BYTE := 0;
	
	s03byte0bit01_res:BYTE := 0;
	s03byte0bit23_water_coller_motor:BYTE := 0;
	s03byte0bit45_cooler_fan:BYTE := 0;
	s03byte0bit67_lowpress_pump:BYTE := 0;
	
	s03byte3bit0_all_wash_sweep:BOOL := FALSE;
	s03byte3bit1_left_wash_sweep:BOOL := FALSE;
	s03byte3bit2_right_wash_sweep:BOOL := FALSE;
	s03byte3bit3_all_sweep:BOOL := FALSE;
	s03byte3bit4_left_sweep:BOOL := FALSE;
	s03byte3bit5_right_sweep:BOOL := FALSE;
	s03byte3bit6_all_wash:BOOL := FALSE;
	s03byte3bit7_left_wash:BOOL := FALSE;
	
	s03byte4bit0_right_wash:BOOL := FALSE;
	s03byte4bit1_stop_sweep:BOOL := FALSE;
	s03byte4bit2_fog_pump:BOOL := FALSE;
	s03byte4bit3_selfclean:BOOL := FALSE;
	s03byte4bit4_boxdoor_close:BOOL := FALSE;
	s03byte4bit5_boxdoor_open:BOOL := FALSE;
	s03byte4bit6_box_up:BOOL := FALSE;
	s03byte4bit7_box_down:BOOL := FALSE;
	
	s03byte5bit0_motor_start:BOOL := FALSE;
	s03byte5bit1_motor_stop:BOOL := FALSE;
	s03byte5bit4_normal_speed:BOOL := FALSE;
	s03byte5bit5_high_speed:BOOL := FALSE;
	s03byte5bit6_sweeper_high_speed:BOOL := FALSE;
	s03byte5bit7_sweeper_middle_spped:BOOL := FALSE;
	
	s03byte6bit0_sweeper_low_speed:BOOL := FALSE;
	s03byte6bit1_highpress_wash:BOOL := FALSE;
	s03byte6bit2_drain_start:BOOL := FALSE;
	s03byte6bit3_drain_auto:BOOL := FALSE;
	s03byte6bit4_drain_manual:BOOL := FALSE;
	s03byte6bit5_drain_left_shooter:BOOL := FALSE;
	s03byte6bit6_drain_right_shooter:BOOL := FALSE;
	s03byte6bit7_sub_drain:BOOL := FALSE;
	
	s03byte7bit0_drain_selfclean:BOOL := FALSE;
	s03byte7bit1_change_sweeper:BOOL := FALSE;
	s03byte7bit2_func_test:BOOL := FALSE;
	s03byte7bit3_intelligent:BOOL := FALSE;
	s03byte7bit4_cleanly:BOOL := FALSE;
	s03byte7bit5_normal:BOOL := FALSE;
	s03byte7bit6_dirty:BOOL := FALSE;
	s03byte7bit7_wastewater_pump:BOOL := FALSE;
	
	s04byte0bit0_point_shoot_up:BOOL := FALSE;
	s04byte0bit1_point_shoot_down:BOOL := FALSE;
	s04byte0bit2_point_shoot_left:BOOL := FALSE;
	s04byte0bit3_point_shoot_right:BOOL := FALSE;
	s04byte0bit4_sucker_shooter_drain:BOOL := FALSE;
	
	s04byte1bit3_test_cooler_motor:BOOL := FALSE;
	s04byte1bit4_test_cooler_fan:BOOL := FALSE;
	s04byte1bit5_test_sweeper_middle:BOOL := FALSE;
	s04byte1bit6_test_sweeper_low:BOOL := FALSE;
	s04byte1bit7_test_left_sweep:BOOL := FALSE;
	
	s04byte2bit0_test_right_sweep:BOOL := FALSE;
	s04byte2bit1_test_all_sweep:BOOL := FALSE;
	s04byte2bit2_test_box_down:BOOL := FALSE;
	s04byte2bit3_test_box_up:BOOL := FALSE;
	s04byte2bit4_test_sucker_down:BOOL := FALSE;
	s04byte2bit5_test_sucker_up:BOOL := FALSE;
	s04byte2bit6_test_boxdoor_open:BOOL := FALSE;
	s04byte2bit7_test_boxdoor_close:BOOL := FALSE;
	
	s04byte3bit0_test_left_sweeper_down:BOOL := FALSE;
	s04byte3bit1_test_left_sweeper_up:BOOL := FALSE;
	s04byte3bit2_test_right_sweeper_down:BOOL := FALSE;
	s04byte3bit3_test_right_sweeper_up:BOOL := FALSE;
	s04byte3bit4_test_left_shooter_out:BOOL := FALSE;
	s04byte3bit5_test_right_shooter_out:BOOL := FALSE;
	s04byte3bit6_test_left_shooter_water:BOOL := FALSE;
	s04byte3bit7_test_right_shooter_water:BOOL := FALSE;
	
	s04byte4bit0_test_sucker_water:BOOL := FALSE;
	s04byte4bit1_test_highpress_wash:BOOL := FALSE;
	s04byte4bit2_test_selfclean:BOOL := FALSE;
	s04byte4bit3_test_highpress_pump_gearin:BOOL := FALSE;
	s04byte4bit4_test_fog_pump:BOOL := FALSE;
	s04byte4bit5_test_left_sweeper_out:BOOL := FALSE;
	s04byte4bit6_test_right_sweeper_out:BOOL := FALSE;
	s04byte4bit7_test_wastewater_pump:BOOL := FALSE;
	
	s04byte5bit0_test_wastewater_valve:BOOL := FALSE;
	s04byte5bit1_test_backup_power:BOOL := FALSE;
	s04byte5bit6_motor_starting:BOOL := FALSE;
	s04byte5bit7_system_running:BOOL := FALSE;
	
	s05byte45_speed_change_value:UINT := 0;
	s05byte67_sub_motor_min_speed:UINT := 0;
	
	s06byte01_normal_speed:UINT := 0;
	s06byte23_high_speed:UINT := 0;
	s06byte45_sweeper_speed:UINT := 0;
	
	s07byte01_highpress_pump_high_speed:UINT := 0;
	s07byte23_highpress_pump_high_speed_stop:UINT := 0;
	s07byte45_sub_motor_max_speed:UINT := 0;
	s07byte67_sub_motor_idle_speed:UINT := 0;
	
	s08byte01_real_torque:UINT := 0;
	s08byte23_real_speed:UINT := 0;
	s08byte45_bus_voltage:UINT := 0;
	s08byte67_phase_current:UINT := 0;
	
	s09byte01_max_dirve_torque:UINT := 0;
	s09byte23_max_brake_torque:UINT := 0;
	s09byte4_temp_controller:BYTE := 0;
	s09byte5_temp_motor:BYTE := 0;
	s09byte67_motor_max_speed:UINT := 0;
	
	s10byte0bit23_direction_cw:BYTE := 0;
	s10byte0bit45_motor_mode:BYTE := 0;
	s10byte0bit67_motor_stat:BYTE := 0;
	
	s10byte1bit01_bus_low_voltage:BYTE := 0;
	s10byte1bit23_bus_high_voltage:BYTE := 0;
	s10byte1bit45_ctrller_high_temp:BYTE := 0;
	s10byte1bit67_motor_high_temp:BYTE := 0;
	
	s10byte2bit01_igbt_fault:BYTE := 0;
	s10byte2bit23_overspeed:BYTE := 0;
	s10byte2bit45_comm_error:BYTE := 0;
	s10byte2bit67_short:BYTE := 0;
	
	s10byte3bit01_motor_overload:BYTE := 0;
	s10byte3bit23_selfcheck_fault:BYTE := 0;
	s10byte3bit45_low_voltage:BYTE := 0;
	s10byte3bit67_sensor_fault:BYTE := 0;
	
	s11byte0_chassis_power_percent:BYTE := 0;
	s11byte1_res :BYTE := 0;
	s11byte23_speed_set_value:UINT := 0;
	s11byte45_version:UINT := 0;
	
	//底盘handle
	hReceiver_ready:CAA.HANDLE;
	hReceiver_speed:CAA.HANDLE;
	hReceiver_soc:CAA.HANDLE;
	
	//显示屏 0x0c00 074f ~ 0x0c04 074f
	hRecver_screen:CAA.HANDLE;
	
	tmp_byte:BYTE;
	tmp_uint:UINT;
	Err:CAA.ERROR;
	
	hMsg : CAA.HANDLE;
	nReceived : CAA.COUNT;
	nAvailable: CAA.COUNT;
	ReadErr   : CAA.ERROR;
	MsgID     : CL2I.COBID;	
	pRxData :POINTER TO CL2I.DATA;
	
	can_stat : DINT := 0;
END_VAR

CASE can_stat OF
	0:   //init can port0 and port1
		hCan0 := cl2.DriverOpenH(usiNetId:=0,uiBaudRate:=250,xSupport29Bits:=TRUE,ctMessages:=100,peError:=ADR(Err));	 //CAN1
		IF hCan0 > 0 THEN
			can_stat := 10;
		END_IF
	
	10: //create receiver for data
		//创建接收底盘信息的接收器: ID:0x18c21726,  byte6.bit2  READY灯	
	  	hReceiver_ready := CL2.CreateMaskReceiver(hDriver := hCan0,
			cobIdValue := 16#18C21726, //cobID value
			cobIdMask := 16#FFFFFFFF, //cobID mask ==> all bits of value are relevant									
			xRTRValue := FALSE, //no RTR messages
			xRTRMask := FALSE, //activate RTR filter ==> xRTRValue will be checked
			x29BitIdValue := TRUE, //29 bit CAN messages
			x29BitIdMask := TRUE, //activate 29 bit filter ==> x29BitIdValue will be checked
			xTransmitValue := FALSE, //only receive messages, no transmit message loopback
			xTransmitMask := FALSE, //activate transmit mask filter ==> xTransmitValue will be checked
			xAlwaysNewest := FALSE, //FALSE := receiver with queue; TRUE: only newest message
			eEvent := CB.EVENT.NO_EVENT,  //no receive event
			xEnableSyncWindow := FALSE, //not implemented
			peError := ADR(Err) //optional pointer to error
			);
		//创建接收底盘信息的接收器: ID:0x18c31726,  byte7  车速	
	  	hReceiver_speed := CL2.CreateMaskReceiver(hDriver := hCan0,
			cobIdValue := 16#18C31726, //cobID value
			cobIdMask := 16#FFFFFFFF, //cobID mask ==> all bits of value are relevant									
			xRTRValue := FALSE, //no RTR messages
			xRTRMask := FALSE, //activate RTR filter ==> xRTRValue will be checked
			x29BitIdValue := TRUE, //29 bit CAN messages
			x29BitIdMask := TRUE, //activate 29 bit filter ==> x29BitIdValue will be checked
			xTransmitValue := FALSE, //only receive messages, no transmit message loopback
			xTransmitMask := FALSE, //activate transmit mask filter ==> xTransmitValue will be checked
			xAlwaysNewest := FALSE, //FALSE := receiver with queue; TRUE: only newest message
			eEvent := CB.EVENT.NO_EVENT, //no receive event
			xEnableSyncWindow := FALSE, //not implemented
			peError := ADR(Err) //optional pointer to error
			);	
		
		//创建接收底盘信息的接收器: ID:0x182126f4,  byte0*0.4  剩余SOC百分比
		hReceiver_soc := CL2.CreateMaskReceiver(hDriver := hCan0,
			cobIdValue := 16#182126F4, //cobID value
			cobIdMask := 16#FFFFFFFF, //cobID mask ==> all bits of value are relevant									
			xRTRValue := FALSE, //no RTR messages
			xRTRMask := FALSE, //activate RTR filter ==> xRTRValue will be checked
			x29BitIdValue := TRUE, //no 29 bit CAN messages
			x29BitIdMask := TRUE, //activate 29 bit filter ==> x29BitIdValue will be checked
			xTransmitValue := FALSE, //only receive messages, no transmit message loopback
			xTransmitMask := FALSE, //activate transmit mask filter ==> xTransmitValue will be checked
			xAlwaysNewest := FALSE, //FALSE := receiver with queue; TRUE: only newest message
			eEvent := CB.EVENT.NO_EVENT, //no receive event
			xEnableSyncWindow := FALSE, //not implemented
			peError := ADR(Err) //optional pointer to error
		);
		//创建接收显示屏信息的接收器: ID:0x0cxx074f
		hRecver_screen := CL2.CreateMaskReceiver(hDriver := hCan0,
			cobIdValue := 16#0C00074F, //cobID value  
			cobIdMask := 16#FFFCFFFF, //cobID mask	0c00074f,0c01074f,0c02074f,0c03074f,							
			xRTRValue := FALSE, //no RTR messages
			xRTRMask := FALSE, //activate RTR filter ==> xRTRValue will be checked
			x29BitIdValue := TRUE, //no 29 bit CAN messages
			x29BitIdMask := TRUE, //activate 29 bit filter ==> x29BitIdValue will be checked
			xTransmitValue := FALSE, //only receive messages, no transmit message loopback
			xTransmitMask := FALSE, //activate transmit mask filter ==> xTransmitValue will be checked
			xAlwaysNewest := FALSE, //FALSE := receiver with queue; TRUE: only newest message
			eEvent := CB.EVENT.NO_EVENT, //no receive event
			xEnableSyncWindow := FALSE, //not implemented
			peError := ADR(Err) //optional pointer to error
		);
		
		IF (hReceiver_ready <> 0 AND hReceiver_speed <> 0 AND hReceiver_soc <> 0 AND hRecver_screen <> 0 ) THEN
			 can_stat := 20;
		ELSE
			RETURN;
		END_IF
	
	20:  //receive data
		//接收底盘信息: ID:0x18c21726,  byte6.bit2  READY灯	
		nReceived := cl2.GetMsgCount(hReceiverId :=hReceiver_ready, peError := ADR(ReadErr));
		IF nReceived <> 0 THEN
			hMsg := cl2.Read(hReceiverId :=hReceiver_ready,pctMsgLeft:=ADR(nAvailable),peError:=ADR(ReadErr));
			pRxData := cl2.GetMessageDataPointer(hMessage:= hMsg,peError:=ADR(ReadErr));	
			tmp_byte := pRxData^[6];
			can_data_ready := tmp_byte.2;
			cl2.FreeMessage(hMsg);
		END_IF

		//接收底盘信息: ID:0x18c31726,  byte7  车速	
		nReceived := cl2.GetMsgCount(hReceiverId :=hReceiver_speed, peError := ADR(ReadErr));
		IF nReceived <> 0 THEN
			hMsg := cl2.Read(hReceiverId :=hReceiver_speed,pctMsgLeft:=ADR(nAvailable),peError:=ADR(ReadErr));
			pRxData := cl2.GetMessageDataPointer(hMessage:= hMsg,peError:=ADR(ReadErr));	
			can_data_speed := pRxData^[6];
			cl2.FreeMessage(hMsg);
		END_IF

		//接收底盘信息: ID:0x182126f4,  byte0*0.4  剩余SOC百分比
		nReceived := cl2.GetMsgCount(hReceiverId :=hReceiver_soc, peError := ADR(ReadErr));
		IF nReceived <> 0 THEN
			hMsg := cl2.Read(hReceiverId :=hReceiver_soc,pctMsgLeft:=ADR(nAvailable),peError:=ADR(ReadErr));
			pRxData := cl2.GetMessageDataPointer(hMessage:= hMsg,peError:=ADR(ReadErr));	
			tmp_uint := ANY_TO_UINT(pRxData^[0]);
			can_data_soc := ANY_TO_BYTE(tmp_uint*2/5);
			cl2.FreeMessage(hMsg);
		END_IF	

		//接收显示屏信息: ID:0x0cXX074f
		nReceived := cl2.GetMsgCount(hReceiverId :=hRecver_screen, peError := ADR(ReadErr));
		IF nReceived <> 0 THEN
			hMsg := cl2.Read(hReceiverId :=hRecver_screen,pctMsgLeft:=ADR(nAvailable),peError:=ADR(ReadErr));
			pRxData := cl2.GetMessageDataPointer(hMessage:= hMsg,peError:=ADR(ReadErr));	
			MsgID := cl2.GetMessageId(hMessage := hMsg, peError := ADR(ReadErr));
			//处理接收数据
			//proc_screen_data(MsgID := MsgID, pRxData := pRxData);
			cl2.FreeMessage(hMsg);
		END_IF
		
		can_stat := 30;
	30:  //send data to screen
		// 12帧数据一起发送，以后可以根据需要调整发送间隔
		
		//填充发送缓冲区
		
		can_stat := 20;

	100:   //error
		
END_CASE

END_PROGRAM

// Changsha_Xiangji_ARM_Cortex_A9_xilinx_zynq7000_linux/Application/CAN_COMM/prg_can1
PROGRAM prg_can1    //CAN1   与上装电机驱动器通信
VAR
	hCan1:CAA.HANDLE:=0;
    CanWriteData : ARRAY[0..7] OF BYTE;
    CanWriteMsgID:UDINT;
	CanReadData : ARRAY[0..7] OF BYTE;  
	CanReadMsgID:UDINT;
	bModifyTimeFlag :BOOL := FALSE;
	
	//通过CAN总线从驱动器读到的信息
	c11byte01_torque:UINT:= 0;
	c11byte23_speed:UINT:= 0;
	c11byte45_voltage:UINT:=0;
	c11byte67_current:UINT:= 0;
	
	c12byte01_drv_torque_max:UINT:= 0;
	c12byte23_brk_torque_max:UINT := 0;
	c12byte4_temp_controller:INT:= 0; //offset:  -40
	c12byte5_temp_motor:INT := 0;  //offset: -40
	c12byte67_speed_max:UINT:= 0;  
	
	c13byte0bit23_cw:BYTE:=0; //00:stop, 01:ccw,  10:cw
	c13byte0bit45_mode:BYTE := 01; //01:drive, 10:brake
	c13byte0bit67_stat:BYTE := 00; //00: enable, 01:running, 10:stop, 11:fault
	
	c13byte1bit01_low_vol:BYTE := 00; //00: normal, 01:warning, 10: fault
	c13byte1bit23_high_vol:BYTE := 0;
	c13byte1bit45_temp_ctrler:BYTE := 0;
	c13byte1bit67_temp_motor:BYTE := 0;
	
	c13byte2bit01_igbt:BYTE := 0;
	c13byte2bit23_speed:BYTE := 0;
	c13byte2bit45_comm:BYTE := 0;
	c13byte2bit67_short:BYTE := 0;
	
	c13byte3bit01_overload:BYTE := 0;
	c13byte3bit23_selfcheck:BYTE := 0;
	c13byte3bit45_low_voltage:BYTE := 0;
	c13byte3bit67_sensor:BYTE := 0;
	
	
	//发送给驱动器的信息
	byte0bit6_enable:BOOL := FALSE;
	byte0bit45_cw:BYTE := 01;  //01:CCW,  10:CW 方向
	byte0bit23_ctrl:BYTE := 01; //01:转矩， 10：转速
	byte0bit01_mode:BYTE := 01;  //01:牵引， 10: 制动
	byte12_torque:UINT:= 0; //转矩
	byte34_speed:UINT := 0;  //转速
	


	hReceiver1:CAA.HANDLE;
	hReceiver2:CAA.HANDLE;
	hReceiver3:CAA.HANDLE;
	tmp_byte:BYTE;
	tmp_uint:UINT;
	Err:CAA.ERROR;
	
	hMsg : CAA.HANDLE;
	nReceived : CAA.COUNT;
	nAvailable: CAA.COUNT;
	ReadErr   : CAA.ERROR;
	MsgID     : CL2I.COBID;	
	pRxData :POINTER TO CL2I.DATA;
	
	can_stat : DINT := 0;
END_VAR

CASE can_stat OF
	0:   //init can port1
		hCan1 := cl2.DriverOpenH(usiNetId:=1,uiBaudRate:=250,xSupport29Bits:=TRUE,ctMessages:=100,peError:=ADR(Err));	 //CAN1
		IF hCan1 > 0 THEN
			can_stat := 10;
		END_IF
	
	10: //create receiver for data
		//接收驱动器信息1: ID:0x0C112AEE,  
	  	hReceiver1 := CL2.CreateMaskReceiver(hDriver := hCan1,
			cobIdValue := 16#0C112AEE, //cobID value
			cobIdMask := 16#FFFFFFFF, //cobID mask ==> all bits of value are relevant									
			xRTRValue := FALSE, //no RTR messages
			xRTRMask := FALSE, //activate RTR filter ==> xRTRValue will be checked
			x29BitIdValue := TRUE, //29 bit CAN messages
			x29BitIdMask := TRUE, //activate 29 bit filter ==> x29BitIdValue will be checked
			xTransmitValue := FALSE, //only receive messages, no transmit message loopback
			xTransmitMask := FALSE, //activate transmit mask filter ==> xTransmitValue will be checked
			xAlwaysNewest := FALSE, //FALSE := receiver with queue; TRUE: only newest message
			eEvent := CB.EVENT.NO_EVENT,  //no receive event
			xEnableSyncWindow := FALSE, //not implemented
			peError := ADR(Err) //optional pointer to error
			);
		//接收驱动器信息2: ID:0x0C122AEE	
	  	hReceiver2 := CL2.CreateMaskReceiver(hDriver := hCan1,
			cobIdValue := 16#0C122AEE, //cobID value
			cobIdMask := 16#FFFFFFFF, //cobID mask ==> all bits of value are relevant									
			xRTRValue := FALSE, //no RTR messages
			xRTRMask := FALSE, //activate RTR filter ==> xRTRValue will be checked
			x29BitIdValue := TRUE, //29 bit CAN messages
			x29BitIdMask := TRUE, //activate 29 bit filter ==> x29BitIdValue will be checked
			xTransmitValue := FALSE, //only receive messages, no transmit message loopback
			xTransmitMask := FALSE, //activate transmit mask filter ==> xTransmitValue will be checked
			xAlwaysNewest := FALSE, //FALSE := receiver with queue; TRUE: only newest message
			eEvent := CB.EVENT.NO_EVENT, //no receive event
			xEnableSyncWindow := FALSE, //not implemented
			peError := ADR(Err) //optional pointer to error
			);	
		
		//接收驱动器信息3: ID:0x0C132AEE
		hReceiver3 := CL2.CreateMaskReceiver(hDriver := hCan1,
			cobIdValue := 16#0C132AEE, //cobID value
			cobIdMask := 16#FFFFFFFF, //cobID mask ==> all bits of value are relevant									
			xRTRValue := FALSE, //no RTR messages
			xRTRMask := FALSE, //activate RTR filter ==> xRTRValue will be checked
			x29BitIdValue := TRUE, //no 29 bit CAN messages
			x29BitIdMask := TRUE, //activate 29 bit filter ==> x29BitIdValue will be checked
			xTransmitValue := FALSE, //only receive messages, no transmit message loopback
			xTransmitMask := FALSE, //activate transmit mask filter ==> xTransmitValue will be checked
			xAlwaysNewest := FALSE, //FALSE := receiver with queue; TRUE: only newest message
			eEvent := CB.EVENT.NO_EVENT, //no receive event
			xEnableSyncWindow := FALSE, //not implemented
			peError := ADR(Err) //optional pointer to error
		);
		IF (hReceiver1 <> 0 AND hReceiver2 <> 0 AND hReceiver3 <> 0 ) THEN
			 can_stat := 20;
		ELSE
			RETURN;
		END_IF
	20:  //send data 
		can1_set_send_buf(ADR(canWriteData));
		CAN_Send_MSG(hCan1, 16#0801EE2A, 8, CanWriteData);
		can_stat := 30;
	
	30:  //receive data
		//接收驱动器信息1: ID:0x0C112AEE,  
		nReceived := cl2.GetMsgCount(hReceiverId :=hReceiver1, peError := ADR(ReadErr));
		IF nReceived <> 0 THEN
			hMsg := cl2.Read(hReceiverId :=hReceiver1,pctMsgLeft:=ADR(nAvailable),peError:=ADR(ReadErr));
			pRxData := cl2.GetMessageDataPointer(hMessage:= hMsg,peError:=ADR(ReadErr));	
			can1_get_data1(pRxData);
			cl2.FreeMessage(hMsg);
		END_IF

		//接收驱动器信息2: ID:0x0C122AEE
		nReceived := cl2.GetMsgCount(hReceiverId :=hReceiver2, peError := ADR(ReadErr));
		IF nReceived <> 0 THEN
			hMsg := cl2.Read(hReceiverId :=hReceiver2,pctMsgLeft:=ADR(nAvailable),peError:=ADR(ReadErr));
			pRxData := cl2.GetMessageDataPointer(hMessage:= hMsg,peError:=ADR(ReadErr));	
			can1_get_data2(pRxData);
			cl2.FreeMessage(hMsg);
		END_IF

		//接收驱动器信息3: ID:0x0C132AEE
		nReceived := cl2.GetMsgCount(hReceiverId :=hReceiver3, peError := ADR(ReadErr));
		IF nReceived <> 0 THEN
			hMsg := cl2.Read(hReceiverId :=hReceiver3,pctMsgLeft:=ADR(nAvailable),peError:=ADR(ReadErr));
			pRxData := cl2.GetMessageDataPointer(hMessage:= hMsg,peError:=ADR(ReadErr));	
			can1_get_data3(pRxData);
			cl2.FreeMessage(hMsg);
		END_IF	
		
		can_stat := 20;
	
	
	100:   //error
		
		
END_CASE

METHOD can1_get_data1 : bool
VAR_INPUT
	pRxData :POINTER TO CL2I.DATA;
END_VAR

VAR
	tmp_byte : BYTE := 0;
	tmp_uint: UINT := 0;
END_VAR
c11byte01_torque := 256*ANY_TO_UINT(pRxData^[1]) + ANY_TO_UINT(pRxData^[0]);
c11byte23_speed :=  256*ANY_TO_UINT(pRxData^[3]) + ANY_TO_UINT(pRxData^[2]);
c11byte45_voltage :=  256*ANY_TO_UINT(pRxData^[5]) + ANY_TO_UINT(pRxData^[4]);
c11byte67_current :=  256*ANY_TO_UINT(pRxData^[7]) + ANY_TO_UINT(pRxData^[6]);

can1_get_data1 := TRUE;
END_METHOD

METHOD can1_get_data3 : bool
VAR_INPUT
	pRxData :POINTER TO CL2I.DATA;
END_VAR

VAR
	tmp_byte : BYTE := 0;
	tmp_uint: UINT := 0;
END_VAR
tmp_byte := pRxData^[0];
c13byte0bit23_cw := ANY_TO_BYTE(tmp_byte.3)*2 + ANY_TO_BYTE(tmp_byte.2);
c13byte0bit45_mode := ANY_TO_BYTE(tmp_byte.5)*2 + ANY_TO_BYTE(tmp_byte.4);
c13byte0bit67_stat := ANY_TO_BYTE(tmp_byte.7)*2 + ANY_TO_BYTE(tmp_byte.6); 

tmp_byte := pRxData^[1];
c13byte1bit01_low_vol := ANY_TO_BYTE(tmp_byte.1)*2 + ANY_TO_BYTE(tmp_byte.0);
c13byte1bit23_high_vol := ANY_TO_BYTE(tmp_byte.3)*2 + ANY_TO_BYTE(tmp_byte.2);
c13byte1bit45_temp_ctrler := ANY_TO_BYTE(tmp_byte.5)*2 + ANY_TO_BYTE(tmp_byte.4);
c13byte1bit67_temp_motor := ANY_TO_BYTE(tmp_byte.7)*2 + ANY_TO_BYTE(tmp_byte.6);

tmp_byte := pRxData^[2];
c13byte2bit01_igbt := ANY_TO_BYTE(tmp_byte.1)*2 + ANY_TO_BYTE(tmp_byte.0);
c13byte2bit23_speed := ANY_TO_BYTE(tmp_byte.3)*2 + ANY_TO_BYTE(tmp_byte.2);
c13byte2bit45_comm := ANY_TO_BYTE(tmp_byte.5)*2 + ANY_TO_BYTE(tmp_byte.4);
c13byte2bit67_short := ANY_TO_BYTE(tmp_byte.7)*2 + ANY_TO_BYTE(tmp_byte.6);

tmp_byte := pRxData^[3];
c13byte3bit01_overload := ANY_TO_BYTE(tmp_byte.1)*2 + ANY_TO_BYTE(tmp_byte.0);
c13byte3bit23_selfcheck := ANY_TO_BYTE(tmp_byte.3)*2 + ANY_TO_BYTE(tmp_byte.2);
c13byte3bit45_low_voltage := ANY_TO_BYTE(tmp_byte.5)*2 + ANY_TO_BYTE(tmp_byte.4);
c13byte3bit67_sensor := ANY_TO_BYTE(tmp_byte.7)*2 + ANY_TO_BYTE(tmp_byte.6);

can1_get_data3 := TRUE;
END_METHOD

METHOD can1_get_data2 : bool
VAR_INPUT
	pRxData :POINTER TO CL2I.DATA;
END_VAR

VAR
	tmp_byte : BYTE := 0;
	tmp_uint: UINT := 0;
END_VAR

c12byte01_drv_torque_max := 256*ANY_TO_UINT(pRxData^[1]) + ANY_TO_UINT(pRxData^[0]);
c12byte23_brk_torque_max := 256*ANY_TO_UINT(pRxData^[3]) + ANY_TO_UINT(pRxData^[2]);
c12byte4_temp_controller := ANY_TO_INT(pRxData^[4]) - 40;
c12byte5_temp_motor := ANY_TO_INT(pRxData^[5]) - 40;
c12byte67_speed_max :=  256*ANY_TO_UINT(pRxData^[7]) + ANY_TO_UINT(pRxData^[6]);

can1_get_data2 := TRUE;
END_METHOD

METHOD can1_set_send_buf : bool
VAR_INPUT
	pData :POINTER TO CL2I.DATA;
END_VAR

VAR
	tmp_byte : BYTE := 0;
END_VAR
tmp_byte := 0;
tmp_byte.6 := byte0bit6_enable;
tmp_byte := tmp_byte + byte0bit45_cw*16;
tmp_byte := tmp_byte + byte0bit23_ctrl*4;
tmp_byte := tmp_byte + byte0bit01_mode*1;

can1_set_send_buf := TRUE;
END_METHOD

END_PROGRAM

// Changsha_Xiangji_ARM_Cortex_A9_xilinx_zynq7000_linux/Application/CAN_COMM/CAN_Send_MSG
FUNCTION CAN_Send_MSG : BOOL
VAR_INPUT
	h:	dword;     //hCan
	TMsgID   : CL2I.COBID;
    TusiLen  : USINT;
	TData    : ARRAY[0..7] OF BYTE;    	
END_VAR
VAR
   Send:CAA.HANDLE;
   WriteErr   : CL2.ERROR;
   p_data:POINTER TO CL2I.DATA;
END_VAR

IF  (0=h) THEN
	RETURN;
END_IF 

Send := cl2.CreateMessage(hDriver := h,
                          cobID := TMsgID,
						  usiLength := TusiLen,
						  xRTR := FALSE,
						  x29BitID := TRUE,
						  peError := ADR(WriteErr));
						  
IF Send <> CAA.gc_hINVALID THEN
	p_data := cl2.GetMessageDataPointer(hMessage := Send,peError:=ADR(WriteErr));
	IF (WriteErr = CL2.ERROR.NO_ERROR) THEN
		SysMemCpy(pDest:=p_data,pSrc:=ADR(TData),udiCount:=SIZEOF(TData));
	END_IF
	
	WriteErr := cl2.Write(hDriver := h,hMessage:=Send,usiPriority:=1,xEnableSyncWindow:=FALSE);
	IF (WriteErr <> CL2.ERROR.NO_ERROR) THEN
        cl2.FreeMessage(hMessage:=Send);		
	END_IF
	
	p_data := CAA.gc_pNULL;
	Send:=CAA.gc_hINVALID;	
END_IF

END_FUNCTION

// Changsha_Xiangji_ARM_Cortex_A9_xilinx_zynq7000_linux/Application/CAN_COMM/prg_test_can
PROGRAM prg_test_can
VAR
	hCan0:CAA.HANDLE:=0;
	hCan1:CAA.HANDLE:=0;
	cmd_test:BOOL := FALSE;
    CanWriteData : ARRAY[0..7] OF BYTE;
    CanWriteMsgID:UDINT;
	CanReadData : ARRAY[0..7] OF BYTE;  
	CanReadMsgID:UDINT;		
	test_01:BOOL := FALSE;
	test_02:BOOL := FALSE;
	test_03:BOOL := FALSE;
	test_04:BOOL := FALSE;
	test_05:BOOL := FALSE;
	test_06:BOOL := FALSE;
	test_07:BOOL := FALSE;
	
END_VAR


IF NOT cmd_test THEN 
	RETURN;
END_IF

hCan0 := prg_can0.hCan0;
hCan1 := prg_can1.hCan1;

IF test_01 THEN
	CanWriteData[0] := 123;
	CanWriteData[1] := 1;
	CanWriteData[6] := 234;
	CAN_Send_MSG(hCan0, 16#0C112AEE, 8, CanWriteData);	
	test_01 := FALSE;
END_IF

IF test_02 THEN
	CAN_Send_MSG(hCan0, 16#0C122AEE, 8, CanWriteData);	
	test_02 := FALSE;
END_IF

IF test_03 THEN
	CAN_Send_MSG(hCan0, 16#0C132AEE, 8, CanWriteData);
	test_03 := FALSE;	
END_IF

IF test_04 THEN
	CAN_Send_MSG(hCan1, 16#18C21726, 8, CanWriteData);
	test_04 := FALSE;	
END_IF

END_PROGRAM

// Changsha_Xiangji_ARM_Cortex_A9_xilinx_zynq7000_linux/Application/main
VISUALIZATION main  // 2x2
END_VISUALIZATION
